// TIA Portal V16 export
// export: Created 2021-07-12T00:42:28.5404023Z, ExportSetting WithDefaults, DisplayName Totally Integrated Automation Portal, DisplayVersion V16 Update 4, DisplayName TIA Portal Version Control Interface, DisplayVersion V16 Update 2, DisplayName TIA Portal Openness, DisplayVersion V16 Update 4, DisplayName STEP 7 Professional, DisplayVersion V16 Update 4, DisplayName STEP 7 Safety, DisplayVersion V16, DisplayName WinCC Advanced, DisplayVersion V16 Update 4
VAR_GLOBAL   // PLC tag table "Default tag table"
   io_a AT %I0.0 : Bool;
   io_b AT %I0.1 : Bool;
END_VAR
VAR_GLOBAL CONSTANT   // user constants
   MAX_RPM : Int := 2800;
END_VAR
